// TIA Portal V15.1 export
// export: Created 2024-06-21T08:41:12.508101Z, ExportSetting WithDefaults, DisplayName Totally Integrated Automation Portal, DisplayVersion V15.1 Update 5, DisplayName TIA Portal Openness, DisplayVersion V15.1 Update 5, DisplayName SINAMICS Startdrive Advanced, DisplayVersion V15.1, DisplayName G130, G150, S120, S150, SINAMICS MV, S210, DisplayVersion V15.1, DisplayName G110M, G120, G120C, G120D, G120P, DisplayVersion V15.1, DisplayName STEP 7 Professional, DisplayVersion V15.1 Update 5, DisplayName STEP 7 Safety, DisplayVersion V15.1, DisplayName WinCC Professional, DisplayVersion V15.1 Update 5, DisplayName SIMATIC Visualization Architect, DisplayVersion V15.1
FUNCTION_BLOCK "LGBColourGroup"   // FB6700, SCL
{ S7_Optimized_Access := 'TRUE' }
VERSION : 0.1
// stored: AutoNumber false, IsIECCheckEnabled false, IsRetainMemResEnabled false, MemoryReserve 100, SetENOAutomatically False, UDAEnableTagReadback false
   VAR_INPUT
      I_TopCoatColour { ExternalAccessible := 'False'; ExternalVisible := 'False'; ExternalWritable := 'False'} : UDInt;   // Top Coat Colour
      I_ColourGroup { ExternalAccessible := 'False'; ExternalVisible := 'False'; ExternalWritable := 'False'} : "ColourGroup";   // High speed value 0-100% / Colour Group
   END_VAR
   VAR_OUTPUT
      O_TopCoatColourLong { ExternalAccessible := 'False'; ExternalVisible := 'False'; ExternalWritable := 'False'} : Int;   // Top Coat Colour short
      O_TopCoatColour { ExternalAccessible := 'False'; ExternalVisible := 'False'; ExternalWritable := 'False'} : Int;   // Top Coat Colour
      O_ColourGroup { ExternalAccessible := 'False'; ExternalVisible := 'False'; ExternalWritable := 'False'} : Int;   // Colour Group
      O_Alarm { ExternalAccessible := 'False'; ExternalVisible := 'False'; ExternalWritable := 'False'} : Bool;   // Top Coat Colour is not configured in a colour group
   END_VAR
   VAR
      Index { ExternalAccessible := 'False'; ExternalVisible := 'False'; ExternalWritable := 'False'} : Int;   // Index for search function
      SubIndex { ExternalAccessible := 'False'; ExternalVisible := 'False'; ExternalWritable := 'False'} : Int;   // SubIndex for search function
      EndSearch { ExternalAccessible := 'False'; ExternalVisible := 'False'; ExternalWritable := 'False'} : Bool;   // End search function
      TopCoatColourLong { ExternalAccessible := 'False'; ExternalVisible := 'False'; ExternalWritable := 'False'} : Int;   // Top Coat Colour
      TopCoatColour { ExternalAccessible := 'False'; ExternalVisible := 'False'; ExternalWritable := 'False'} : Int;   // Top Coat Colour
      ColourGroup { ExternalAccessible := 'False'; ExternalVisible := 'False'; ExternalWritable := 'False'} : Int;   // Colour Group
      Alarm { ExternalAccessible := 'False'; ExternalVisible := 'False'; ExternalWritable := 'False'} : Bool;   // Top Coat Colour is not configured in a colour group
   END_VAR
BEGIN
   // INIT
   #ColourGroup := 0;
   #TopCoatColour := 0;
   #TopCoatColourLong := 0;
   #Alarm := False;

   // LOGIC
   IF (#I_TopCoatColour < 1000) THEN
       #TopCoatColour := UDINT_TO_INT(#I_TopCoatColour);
   ELSIF (#I_TopCoatColour > 1000) AND (#I_TopCoatColour < 2000) THEN
       #TopCoatColour := UDINT_TO_INT(#I_TopCoatColour) - 1000;
   ELSIF (#I_TopCoatColour > 2000) AND (#I_TopCoatColour < 3000) THEN
       #TopCoatColour := UDINT_TO_INT(#I_TopCoatColour) - 2000;
   ELSIF (#I_TopCoatColour > 9000) AND (#I_TopCoatColour < 10000) THEN
       #TopCoatColour := UDINT_TO_INT(#I_TopCoatColour) - 9000;
   END_IF;

   #Index := 1;
   #EndSearch := False;
   WHILE (#Index <= 5) AND (#TopCoatColour <> 0) AND NOT #EndSearch DO
       #SubIndex := 1;
       WHILE (#SubIndex <= 15) AND (#TopCoatColour <> 0) AND NOT #EndSearch DO
           IF (#TopCoatColour = #I_ColourGroup.ColourGroup[#Index].TopCoatColour[#SubIndex]) THEN
               #ColourGroup := #Index;
               #TopCoatColourLong := UDINT_TO_INT(#I_TopCoatColour);
               #EndSearch := True;
           END_IF;
           #SubIndex := #SubIndex + 1;
       END_WHILE;
       IF (#Index >= 5) AND (#SubIndex > 15) THEN
           #Alarm := True;
           #TopCoatColour := 0;
       END_IF;
       #Index := #Index + 1;
   END_WHILE;

   // OUTPUT
   #O_TopCoatColour := #TopCoatColour;
   #O_TopCoatColourLong := #TopCoatColourLong;
   #O_ColourGroup := #ColourGroup;
   #O_Alarm := #Alarm;
END_FUNCTION_BLOCK
